FUNCTION_BLOCK FB_FormingBoardSpeedControl
VAR_INPUT
    //==============================================================
    // ─────────────── MODE SELECTION / REFERENCES ───────────────
    //==============================================================
    groupSpeedAutoMan          : BOOL;  // TRUE = Auto, FALSE = Manual
    groupAutoSpeedMPM          : REAL;  // Auto speed reference [m/min]
    groupManualSpeedMPM        : REAL;  // Manual speed reference [m/min]
    groupRecoverSpeedCmd       : BOOL;  // Recover (temporary speed bump)
    groupRecoverIncrement      : REAL;  // Recover increment [m/min]
//    interGroupGearRatio        : REAL;  // Inter-group ratio (next section sync)
	paperPresenceSensor				: BOOL;

    tractionRollToSuctionRollGearRatio  : REAL := 0.915;

    //==============================================================
    // ─────────────── DIAMETERS (mm) ───────────────
    //==============================================================
    tractionRollDiameter       : REAL;  // Diameter of group 1 master
    suctionRollDiameter       : REAL;  // Diameter of group 1 slave 1


    //==============================================================
    // ─────────────── CONFIGURATION / LIMITS ───────────────
    //==============================================================
    groupMasterMaxSpeedRPM     : REAL;  // Max allowed master RPM
    rampUpRate					: REAL := 0.1;  // Ramp slow acceleration [RPM/s]
    rampDownRate				: REAL := 0.1;  // Ramp slow acceleration [RPM/s]
	
    rampUpRate2					: REAL := 0.1;  // Ramp fast acceleration [RPM/s]
    rampDownRate2				: REAL := 0.1;  // Ramp fast acceleration [RPM/s]	
	
    state                      : INT;   // Machine state (5 = STOPPING)

	speedDifIncPerPulse		: REAL := 0.05;
	
    groupSpeedDifInc           : BOOL;  // Increment group speed offset
    groupSpeedDifDec           : BOOL;  // Decrement group speed offset
    groupSpeedDifLimLow        : REAL;  // Min offset [%]
    groupSpeedDifLimHigh       : REAL;  // Max offset [%]


    rampReset                  : BOOL;  // Reset ramp command
	
END_VAR


VAR_OUTPUT
    //==============================================================
    // ─────────────── FINAL DRIVE SPEEDS (RPM) ───────────────
    //==============================================================
    tractionRollSpeedRefRPM    : REAL; //Master speed
    suctionRollSpeedRefRPM    : REAL; // Slave speed

    //==============================================================
    // ─────────────── SURFACE SPEEDS (MPM) ───────────────
    //==============================================================
    tractionRollSpeedRefMPM       : REAL;
    suctionRollSpeedRefMPM       : REAL;


    //==============================================================
    // ─────────────── HANDOFF TO NEXT GROUP ───────────────
    //==============================================================
    nextGroupSpeedRefMPM       : REAL;
	speedDif					: REAL;
	
	
	
END_VAR


VAR
    //==============================================================
    // ─────────────── INTERNAL CALCULATION VARIABLES ───────────────
    //==============================================================
    masterMaxSpeedMPM          : REAL;
    baseCmdSpeedMPM            : REAL;
    cmdSpeedMPM                : REAL;
    targetRPM                  : REAL;
    rampTargetRPM              : REAL;
    baseMasterRefRPM           : REAL;
    groupSpeedOffset           : REAL;
    groupDeltaRatioAll         : REAL;
    upperLowerBiasRatio        : REAL;
    useRamp                    : BOOL;
    epsDiameter                : REAL := 0.001;

    // Gear ratios (set externally or calculated elsewhere)


    // Function blocks
    instFB_Gen_SRamp           : FB_Gen_SRamp;
    instFB_SpeedDif_SRamp           : FB_Gen_SRamp;

	rampActive: BOOL;
END_VAR


VAR PERSISTENT
	
    instTUNE2_GroupSpeedDiff   : TUNE2;

END_VAR

//==============================================================
// IMPLEMENTATION
//==============================================================

//====================================================================
// ═══ CALL METHOD TO CALCULATE DIAMETER RATIOS ═════════════════════
//====================================================================
_CalculateGearRatios();

//--------------------------------------------------------------
// Calculate master max surface speed [m/min]
//--------------------------------------------------------------
masterMaxSpeedMPM := groupMasterMaxSpeedRPM * (PI * tractionRollDiameter) / 1000.0;


//--------------------------------------------------------------
// Determine base speed source (auto/manual) + Recover bump
//--------------------------------------------------------------
IF groupSpeedAutoMan THEN
    baseCmdSpeedMPM := groupAutoSpeedMPM;
ELSE
    baseCmdSpeedMPM := groupManualSpeedMPM;
END_IF;

IF groupRecoverSpeedCmd THEN
    cmdSpeedMPM := baseCmdSpeedMPM + groupRecoverIncrement;
ELSE
    cmdSpeedMPM := baseCmdSpeedMPM;
END_IF;


//--------------------------------------------------------------
// Convert MPM → target RPM for the master
//--------------------------------------------------------------
targetRPM := _Scale(
    X    := cmdSpeedMPM,
    I_LO := 0.0,
    I_HI := masterMaxSpeedMPM,
    O_LO := 0.0,
    O_HI := groupMasterMaxSpeedRPM);


//--------------------------------------------------------------
// Ramp handling
//--------------------------------------------------------------
IF state = 5 OR state = 0 THEN
    // STOPPING — force ramp down to zero speed
    rampTargetRPM := 0.0;

ELSIF state = 10 THEN
    // FAULT — clear ramp immediately to ensure no residual motion
    rampTargetRPM := 0.0;
//    rampReset     := TRUE;

ELSE
    // Normal operation — ramp follows target speed
    rampTargetRPM := targetRPM;
//    rampReset     := FALSE;
END_IF;

// Detect when a new target speed change requires ramping
IF paperPresenceSensor THEN
 
  rampActive := TRUE; // Rising edge — ramp request detected

ELSE
	
  rampActive := FALSE; // Rising edge — ramp request detected
  
END_IF;



IF 	paperPresenceSensor THEN
	//slow	
	instFB_Gen_SRamp.A_UP := MAX(0.0, rampUpRate);
	instFB_Gen_SRamp.A_DN := -MAX(0.0, rampDownRate);

ELSE
	//fast
	instFB_Gen_SRamp.A_UP := MAX(0.0, rampUpRate2);
	instFB_Gen_SRamp.A_DN := -MAX(0.0, rampDownRate2);

END_IF


// Ramp function block execution
instFB_Gen_SRamp(
    X          := rampTargetRPM,
//    A_UP       := MAX(0.0, rampUpRate),
//    A_DN       := -MAX(0.0, rampDownRate),
    VU_MAX     := 1000.0,
    VD_MAX     := -1000.0,
    LIMIT_HIGH := groupMasterMaxSpeedRPM,
    RST        := rampReset);

// If ramping, update the baseMasterRefRPM from ramp output
IF rampActive THEN
    baseMasterRefRPM := instFB_Gen_SRamp.Y;

    // Automatically reset ramp flag when the ramp output reaches the target
    IF ABS(instFB_Gen_SRamp.Y - rampTargetRPM) <= 0.05 THEN
//        rampActive := FALSE; // Ramp complete
;
    END_IF;

ELSE
    // No ramping required — direct assignment
    baseMasterRefRPM := rampTargetRPM;
END_IF;


//--------------------------------------------------------------
// Operator offset (TUNE2 control)
//--------------------------------------------------------------
instTUNE2_GroupSpeedDiff(
    SET     := FALSE,
    SU      := groupSpeedDifInc,
    SD      := groupSpeedDifDec,
    RST     := FALSE,
    SS      := speedDifIncPerPulse,
    FS      := speedDifIncPerPulse,
    LIMIT_L := groupSpeedDifLimLow,
    LIMIT_H := groupSpeedDifLimHigh);
//    Y       => groupSpeedOffset);


// Ramp function block execution
instFB_SpeedDif_SRamp(
    X          := instTUNE2_GroupSpeedDiff.Y,
    A_UP       := MAX(0.0, 0.01),
    A_DN       := -MAX(0.0, 0.01),
    VU_MAX     := 1000.0,
    VD_MAX     := -1000.0,
    LIMIT_HIGH := groupSpeedDifLimHigh,
	LIMIT_LOW := groupSpeedDifLimLow,
    RST        := FALSE,
	Y => groupSpeedOffset);

	
speedDif := groupSpeedOffset;
	
groupDeltaRatioAll  := 1.0 + (groupSpeedOffset * 0.01);


//--------------------------------------------------------------
// Apply offsets + calculate all drive RPM references
//--------------------------------------------------------------
tractionRollSpeedRefRPM := baseMasterRefRPM * groupDeltaRatioAll;
suctionRollSpeedRefRPM := tractionRollSpeedRefRPM * tractionRollToSuctionRollGearRatio;


//--------------------------------------------------------------
// Convert RPM → MPM (surface speeds)
//--------------------------------------------------------------
tractionRollSpeedRefMPM := tractionRollSpeedRefRPM * tractionRollDiameter * PI / 1000.0;
suctionRollSpeedRefMPM := (suctionRollSpeedRefRPM * suctionRollDiameter * PI / 1000.0);



//--------------------------------------------------------------
// Suggest downstream handoff (group2 master surface speed)
//--------------------------------------------------------------
nextGroupSpeedRefMPM := tractionRollSpeedRefMPM;


//====================================================================
// ═══ PRIVATE METHOD — CALCULATE DIAMETER RATIOS ════════════════════
//====================================================================
METHOD PRIVATE _CalculateGearRatios
VAR_INPUT
END_VAR
END_METHOD

METHOD PRIVATE _Scale : REAL
VAR_INPUT
    X    : REAL;
    I_LO : REAL;
    I_HI : REAL;
    O_LO : REAL;
    O_HI : REAL;
END_VAR
IF I_LO = I_HI THEN
	_Scale := O_LO;
ELSE
	_Scale := (O_HI - O_LO) / (I_HI - I_LO) * (LIMIT(I_LO, X, I_HI) - I_LO) + O_LO;
END_IF;
END_METHOD

END_FUNCTION_BLOCK

(* stored: Version 1.1.0.1, ProductVersion 3.1.4024.15
   POU FB_FormingBoardSpeedControl: Id {fbd9ef71-4cca-4373-b3e2-d5424b16f9a6}, SpecialFunc None
   Method _CalculateGearRatios: Id {20e3f292-80ac-4748-88f6-514f8f46bf49}
   Method _Scale: Id {2bc9a955-bf28-4083-be2e-7ad292b8142e} *)
